FUNCTION_BLOCK ActivityIndicator EXTENDS HardwareObservationBase
VAR_INPUT
END_VAR
VAR_OUTPUT
END_VAR
VAR
	DO_indic AT%Q*: BOOL;
	
	
	m_sigVar: UINT;
	m_sigState: BOOL;
END_VAR

//FB_Init is always available implicitly and it is used primarily for initialization.
//The return value is not evaluated. For a specific influence, you can also declare the
//methods explicitly and provide additional code there with the standard initialization
//code. You can evaluate the return value.
METHOD FB_Init: BOOL
VAR_INPUT
    bInitRetains: BOOL; // TRUE: the retain variables are initialized (reset warm / reset cold)
    bInCopyCode: BOOL;  // TRUE: the instance will be copied to the copy code afterward (online change)
	
	i_signalProcVar: UINT;
END_VAR
m_sigVar := i_signalProcVar;
END_METHOD

METHOD FlipIndicator : BOOL
VAR_INPUT
END_VAR
m_sigState := FALSE;
DO_indic := NOT DO_indic;
END_METHOD

METHOD  ResetDefinition : BOOL
VAR_INPUT
END_VAR
m_sigState := TRUE;
END_METHOD

METHOD ResetDoneSignal : BOOL
IF m_sigVar = 0 THEN
	ResetDoneSignal := FALSE;
ELSE
	m_sigState  := FALSE;
	ResetDoneSignal := TRUE;
	DO_indic := FALSE;
END_IF
END_METHOD

(*
	Sets the global variable for the "Done" signal to TRUE.
	WIll be reset FlipIndicator is called the next time.
*)
METHOD SetDoneSignal : BOOL
IF m_sigVar = 0 THEN
	SetDoneSignal := FALSE;
ELSE
	m_sigState  := TRUE;
	SetDoneSignal := TRUE;
	DO_indic := FALSE;
END_IF
END_METHOD

(* Update an instance of ProcessState with the part of the process that can be observed by this Hardware Interface. *)
METHOD UpdateProcessObservation : BOOL
VAR_IN_OUT
	io_processState: ProcessState;
END_VAR
io_processState.UpdateState_Binary(m_sigVar, m_sigState, i_force := TRUE);
io_processState.UpdateState_Defined(m_sigVar, TRUE);
END_METHOD

END_FUNCTION_BLOCK

(* stored: Version 1.1.0.1
   POU ActivityIndicator: Id {fc0acb11-6196-4410-a362-9beb79765b3f}, SpecialFunc None
   Method FB_init: Id {fee9e128-cc88-404f-a848-a4f328aea5a4}
   Method FlipIndicator: Id {ebe86216-9bfa-490d-a0c0-08b84d241d97}
   Method ResetDefinition: Id {e22c59ad-cbe5-487a-b192-d96df39e56ad}
   Method ResetDoneSignal: Id {95b734b2-e5f3-4897-80b5-680931ea816a}
   Method SetDoneSignal: Id {58314ac0-973b-40f5-b372-560314e1af36}
   Method UpdateProcessObservation: Id {24c2b38d-f4ff-4734-9150-fdf84dad5fad} *)
